// UDT_Recipe_Processes - Receptová struktura podle procesů
// Tato UDT obsahuje všechny učitelné parametry motorů pro každý proces
// Výchozí hodnoty jsou navrhované - uprav podle stroje

TYPE UDT_Recipe_Processes :
STRUCT
  // Proces: Polohování stolu 1 (Table 1 Positioning) - Servo V90_A1
  Table1_Positioning : STRUCT
    Pos : ARRAY[1..8] OF DINT := [0, 1000, 2000, 3000, 4000, 5000, 6000, 7000];  // Pozice bodů (mm)
    Speed : ARRAY[1..8] OF INT := [100, 200, 300, 400, 500, 400, 300, 200];  // Rychlosti (mm/s)
    Accel : ARRAY[1..8] OF INT := [1000, 1500, 2000, 2500, 3000, 2500, 2000, 1500];  // Akcelerace
  END_STRUCT;

  // Proces: Skenování rotačního hřídele (Rotary Shaft Scanning) - Servo V90_A2
  Rotary_Shaft_Scanning : STRUCT
    Pos : ARRAY[1..8] OF DINT := [0, 45, 90, 135, 180, 225, 270, 315];  // Pozice úhlů (°)
    Speed : ARRAY[1..8] OF INT := [50, 100, 150, 200, 150, 100, 50, 50];  // Rychlosti (°/s)
    Accel : ARRAY[1..8] OF INT := [500, 1000, 1500, 2000, 1500, 1000, 500, 500];  // Akcelerace
  END_STRUCT;

  // Proces: Lepení Z-osa (Gluing Z-Axis) - Servo V90_A3
  Gluing_Z_Axis : STRUCT
    Pos : ARRAY[1..6] OF DINT := [0, 100, 200, 300, 400, 500];  // Pozice (mm)
    Speed : ARRAY[1..6] OF INT := [10, 20, 50, 80, 100, 80];  // Rychlosti (mm/s) - nízké pro lepení
    Accel : ARRAY[1..6] OF INT := [500, 800, 1000, 1200, 1000, 800];  // Akcelerace
  END_STRUCT;

  // Proces: Polohování stolu 2 (Table 2 Positioning) - Servo V90_A4
  Table2_Positioning : STRUCT
    Pos : ARRAY[1..8] OF DINT := [0, 1000, 2000, 3000, 4000, 5000, 6000, 7000];  // Pozice (mm)
    Speed : ARRAY[1..8] OF INT := [100, 200, 300, 400, 500, 400, 300, 200];  // Rychlosti (mm/s)
    Accel : ARRAY[1..8] OF INT := [1000, 1500, 2000, 2500, 3000, 2500, 2000, 1500];  // Akcelerace
  END_STRUCT;

  // Proces: Lineární osa 1 (Linear Axis 1) - IAI_A1
  Linear_Axis1 : STRUCT
    Pos : ARRAY[1..10] OF LREAL := [0.0, 100.0, 200.0, 300.0, 400.0, 500.0, 600.0, 700.0, 800.0, 900.0];  // Pozice (mm)
    Speed : ARRAY[1..10] OF LREAL := [50.0, 100.0, 150.0, 200.0, 250.0, 300.0, 250.0, 200.0, 150.0, 100.0];  // Rychlosti (mm/s)
    Accel : ARRAY[1..10] OF LREAL := [1000.0, 1500.0, 2000.0, 2500.0, 3000.0, 2500.0, 2000.0, 1500.0, 1000.0, 500.0];  // Akcelerace
  END_STRUCT;

  // Proces: Lineární osa 2 (Linear Axis 2) - IAI_A2
  Linear_Axis2 : STRUCT
    Pos : ARRAY[1..10] OF LREAL := [0.0, 80.0, 160.0, 240.0, 320.0, 400.0, 480.0, 560.0, 640.0, 720.0];  // Pozice (mm)
    Speed : ARRAY[1..10] OF LREAL := [50.0, 100.0, 150.0, 200.0, 250.0, 200.0, 150.0, 100.0, 50.0, 50.0];  // Rychlosti (mm/s)
    Accel : ARRAY[1..10] OF LREAL := [1000.0, 1500.0, 2000.0, 2500.0, 2000.0, 1500.0, 1000.0, 500.0, 500.0, 500.0];  // Akcelerace
  END_STRUCT;

  // Proces: Lineární osa 3 (Linear Axis 3) - IAI_A3
  Linear_Axis3 : STRUCT
    Pos : ARRAY[1..10] OF LREAL := [0.0, 60.0, 120.0, 180.0, 240.0, 300.0, 360.0, 420.0, 480.0, 540.0];  // Pozice (mm)
    Speed : ARRAY[1..10] OF LREAL := [20.0, 50.0, 80.0, 100.0, 120.0, 150.0, 120.0, 100.0, 80.0, 50.0];  // Rychlosti (mm/s)
    Accel : ARRAY[1..10] OF LREAL := [500.0, 1000.0, 1500.0, 2000.0, 1500.0, 1000.0, 500.0, 500.0, 500.0, 500.0];  // Akcelerace
  END_STRUCT;

  // Proces: Robot 1 manipulace (Robot 1 Handling) - KukaRobot1
  Robot1_Handling : STRUCT
    Pos : ARRAY[1..20] OF STRUCT(X : LREAL; Y : LREAL; Z : LREAL; A : LREAL; B : LREAL; C : LREAL) := [(0.0,0.0,0.0,0.0,0.0,0.0), ...];  // Kartézské pozice
    Speed : ARRAY[1..20] OF LREAL := [100.0, 150.0, 200.0, 250.0, 300.0, ...];  // Rychlosti (mm/s)
    Accel : ARRAY[1..20] OF LREAL := [500.0, 800.0, 1000.0, 1200.0, 1500.0, ...];  // Akcelerace
  END_STRUCT;

  // Proces: Robot 2 manipulace (Robot 2 Handling) - KukaRobot2
  Robot2_Handling : STRUCT
    Pos : ARRAY[1..20] OF STRUCT(X : LREAL; Y : LREAL; Z : LREAL; A : LREAL; B : LREAL; C : LREAL) := [(0.0,0.0,0.0,0.0,0.0,0.0), ...];  // Kartézské pozice
    Speed : ARRAY[1..20] OF LREAL := [100.0, 150.0, 200.0, 250.0, 300.0, ...];  // Rychlosti (mm/s)
    Accel : ARRAY[1..20] OF LREAL := [500.0, 800.0, 1000.0, 1200.0, 1500.0, ...];  // Akcelerace
  END_STRUCT;

  // Proces: Robot 3 manipulace (Robot 3 Handling) - KukaRobot3
  Robot3_Handling : STRUCT
    Pos : ARRAY[1..20] OF STRUCT(X : LREAL; Y : LREAL; Z : LREAL; A : LREAL; B : LREAL; C : LREAL) := [(0.0,0.0,0.0,0.0,0.0,0.0), ...];  // Kartézské pozice
    Speed : ARRAY[1..20] OF LREAL := [100.0, 150.0, 200.0, 250.0, 300.0, ...];  // Rychlosti (mm/s)
    Accel : ARRAY[1..20] OF LREAL := [500.0, 800.0, 1000.0, 1200.0, 1500.0, ...];  // Akcelerace
  END_STRUCT;

  // Proces: Motor 1 pohyby (Motor 1 Movements) - Motor1
  Motor1_Movements : STRUCT
    Pos : ARRAY[1..17] OF DINT := [0, 1000, 2000, 3000, 4000, 5000, 6000, 7000, 8000, 9000, 10000, 9000, 8000, 7000, 6000, 5000, 4000];  // Pozice
    Speed : ARRAY[1..17] OF INT := [100, 200, 300, 400, 500, 600, 700, 800, 900, 1000, 900, 800, 700, 600, 500, 400, 300];  // Rychlosti
    Accel : ARRAY[1..17] OF INT := [500, 800, 1000, 1200, 1500, 1800, 2000, 1800, 1500, 1200, 1000, 800, 600, 500, 400, 300, 200];  // Akcelerace
  END_STRUCT;

  // Proces: Stopper pohyby (Stopper Movements) - Stopper
  Stopper_Movements : STRUCT
    Pos : ARRAY[1..4] OF DINT := [0, 50, 100, 150];  // Pozice (mm)
    Speed : ARRAY[1..4] OF INT := [50, 100, 150, 200];  // Rychlosti (mm/s)
    Accel : ARRAY[1..4] OF INT := [500, 800, 1000, 1200];  // Akcelerace
  END_STRUCT;

  // Obecné parametry pro všechny procesy
  General_Params : STRUCT
    Homing_Speed : INT := 100;  // Homing rychlost (mm/s nebo °/s)
    Jog_Speed_Plus : INT := 50;  // Jog rychlost +
    Jog_Speed_Minus : INT := 50;  // Jog rychlost -
    Timeout : TIME := T#5S;  // Časový limit pohybu
    Tolerance : LREAL := 0.5;  // Tolerance dosažení pozice (mm/°)
  END_STRUCT;
END_STRUCT;
END_TYPE